INTERFACE I_Logging

METHOD PUBLIC M_Attach : BOOL
VAR_INPUT
	iLogging:				I_Logging;
END_VAR
END_METHOD

METHOD PUBLIC M_Log : BOOL
VAR_INPUT
	eLogLevel:			E_LogLevel;
	nID:				UDINT;
	sSource:			STRING(255);
	sMessage:			STRING(255);
	sArguments:			STRING(255);
END_VAR
END_METHOD

END_INTERFACE

(* stored: Version 1.1.0.1
   Itf I_Logging: Id {8d10f800-b621-4e55-9c3b-f2a551bf051a}
   Method M_Attach: Id {246fd3da-f4e3-4f73-a14a-612d68e14b33}
   Method M_Log: Id {3bf5264c-77ea-40c4-942b-0eebcecbddb2} *)
